// TIA Portal V17 export
// export: Created 2024-01-30T08:49:14.2309531Z, ExportSetting WithDefaults, DisplayName Totally Integrated Automation Portal, DisplayVersion V17 Update 6, DisplayName TIA Portal Openness, DisplayVersion V17 Update 6, DisplayName TIA Portal Version Control Interface, DisplayVersion V17, DisplayName STEP 7 Professional, DisplayVersion V17 Update 6, DisplayName STEP 7 Safety, DisplayVersion V17 Update 6, DisplayName WinCC Advanced, DisplayVersion V17 Update 6
DATA_BLOCK "Festo_ClampingTorque_DB"   // DB15
AUTHOR : Festo SE & Co. KG
FAMILY : Drives
VERSION : 1.0
// stored: AutoNumber true, DBAccessibleFromOPCUA true, DBAccessibleFromWebserver true, InstanceOfName Festo_ClampingTorque, InstanceOfType FB
"Festo_ClampingTorque"
   // VAR_INPUT
   //    Execute : Bool;
   //    LinearRotative : Bool;
   //    ClampingTorque : Real;
   //    PercentForce : USInt;
   //    MAP_HardwareId : HW_IO;
   // END_VAR
   // VAR_OUTPUT
   //    Done : Bool;
   //    Busy : Bool;
   //    Error : Bool;
   //    ErrorId : DWord;
   //    ErrorString : String[50];
   //    ActClampingTorque : Real;
   // END_VAR
   // VAR
   //    ValueWriteREAL { ExternalAccessible := 'False'; ExternalVisible := 'False'; ExternalWritable := 'False'} : Real;
   //    x { ExternalAccessible := 'False'; ExternalVisible := 'False'; ExternalWritable := 'False'} : Real;
   //    Festo_PNU_RW_Single_Instance { S7_SetPoint := 'True'} : "Festo_PNU_RW_Single";
   //    iStep { S7_SetPoint := 'True'} : Int;
   //    iPNU : Int;
   //    udGearEnumerator : UDInt;
   //    udGearDenumerator : UDInt;
   //    xReadWrite : Bool;
   //    xStartParam : Bool;
   //    xBusyParam : Bool;
   //    xDoneParam : Bool;
   //    xErrorParam : Bool;
   //    dwErrorIDParam : DWord;
   //    lValueReadLint : LInt;
   //    rValueReadReal : Real;
   //    rNominalTorque : Real;
   //    rGearFactor : Real;
   //    rTorqueFactor : Real;
   //    trExecuteTrigger : R_TRIG;
   // END_VAR
BEGIN
END_DATA_BLOCK
